{attribute addProperty BoxType "EKM1101-0000-0016"}
{attribute addProperty Id "Up_Out_OFFBIT10.1251"}
{attribute addProperty CRC "615067684"}
{attribute addProperty SizeInBites "16"}
{attribute addProperty SizeInBytes "2"}
TYPE Control_24A93024 :
STRUCT
	{attribute addProperty Name "Up_Out_OFF"}
	Up_Out_OFF : BOOL;
	{attribute 'hide'}
	reserve_1_BIT_0 : BOOL;
	{attribute 'hide'}
	reserve_1_BIT_1 : BOOL;
	{attribute 'hide'}
	reserve_1_BIT_2 : BOOL;
	{attribute 'hide'}
	reserve_1_BIT_3 : BOOL;
	{attribute 'hide'}
	reserve_1_BIT_4 : BOOL;
	{attribute 'hide'}
	reserve_1_BIT_5 : BOOL;
	{attribute 'hide'}
	reserve_1_BIT_6 : BOOL;
	{attribute 'hide'}
	reserve_1_BIT_7 : BOOL;
	{attribute 'hide'}
	reserve_1_BIT_8 : BOOL;
	{attribute 'hide'}
	reserve_1_BIT_9 : BOOL;
	{attribute 'hide'}
	reserve_1_BIT_10 : BOOL;
	{attribute 'hide'}
	reserve_1_BIT_11 : BOOL;
	{attribute 'hide'}
	reserve_1_BIT_12 : BOOL;
	{attribute 'hide'}
	reserve_1_BIT_13 : BOOL;
	{attribute 'hide'}
	reserve_1_BIT_14 : BOOL;
END_STRUCT
END_TYPE

(* stored: Version 1.2.0.0, ProductVersion 3.1.4024.9
   DUT Control_24A93024: Id {e8b3373f-d7b0-45ae-8318-bac1fc5bc6fa} *)
